// Mitsubishi GX Works2 project: TIMER3   PLC: Q03UDV

PROGRAM MAIN
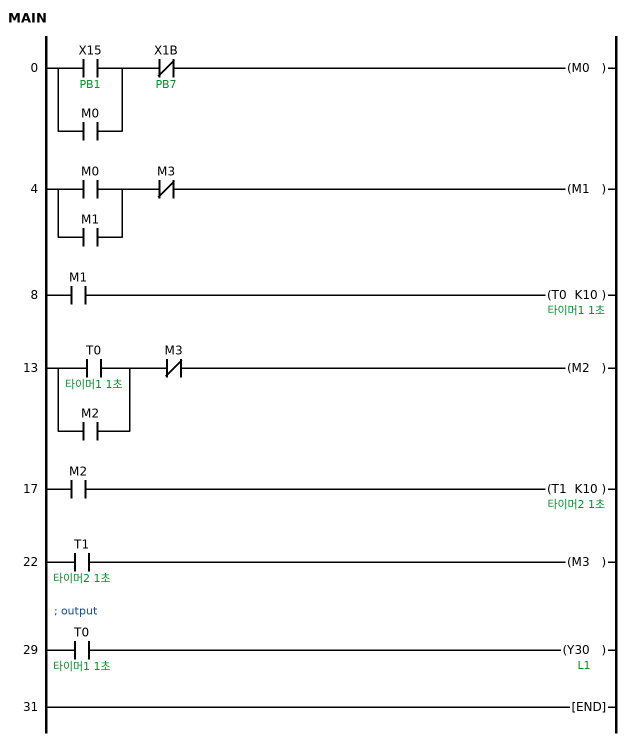
0     LD      X15  ; PB1
      OR      M0
      ANI     X1B  ; PB7
      OUT     M0
4     LD      M0
      OR      M1
      ANI     M3
      OUT     M1
8     LD      M1
      OUT     T0 K10  ; 타이머1 1초
13    LD      T0  ; 타이머1 1초
      OR      M2
      ANI     M3
      OUT     M2
17    LD      M2
      OUT     T1 K10  ; 타이머2 1초
22    LD      T1  ; 타이머2 1초
      OUT     M3
; output
29    LD      T0  ; 타이머1 1초
      OUT     Y30  ; L1
31    END
END_PROGRAM
